// TIA Portal V19 export
TYPE "UDT_CONTROLVALVE"
   STRUCT
      pid : Struct   // PID
         mode { S7_SetPoint := 'True'} : Bool := false;   // Auto=0, Man=1
         action { S7_SetPoint := 'True'} : Bool := false;   // Reverse=0, Forward=1
         spsource : Bool := false;   // 0=internal setpoint, 1=external setpoint
         followup : Bool := false;   // 0=motor control from PID, 1=motor setpoint directly from program
         cmdrst : Bool := false;   // Controller reset command
         pidrun : Bool := false;   // Controller is running
         P { S7_SetPoint := 'True'} : Real := 0.0;   // Proportional gain
         I { S7_SetPoint := 'True'} : DInt := 0;   // Integral action
         D { S7_SetPoint := 'True'} : DInt := 0;   // Derivative action
         SP { S7_SetPoint := 'True'} : Real := 0.0;   // Setpoint
         PV : Real := 0.0;   // Peripheral value
         OFFVAL { S7_SetPoint := 'True'} : Real := 0.0;   // Value loaded to OP when the actuator is stopped
         LMN : Real := 0.0;   // Output of the PID controller
         OP { S7_SetPoint := 'True'} : Real := 0.0;   // Final output to the element
         L { S7_SetPoint := 'True'} : Real := 0.0;   // Lower value
         H { S7_SetPoint := 'True'} : Real := 0.0;   // Higher value
         EXT_SP : Real := 0.0;   // External setpoint
         FUP : Real := 0.0;   // Follow up value
         ITLVAL { S7_SetPoint := 'True'} : Real := 0.0;   // Controller initialization value
         pvunit { S7_SetPoint := 'True'} : WString := WSTRING#'';   // PV Unit
         outunit { S7_SetPoint := 'True'} : WString := WSTRING#'';   // Output Unit
         init : Struct   // Controller initialization routine
            req : Bool := false;   // An initialization routine is required
            dur { S7_SetPoint := 'True'} : Real := 0.0;   // Initialization duration
            delay : "UDT_DELAYON";
         END_STRUCT;
      END_STRUCT;
      unscale : Struct   // Scale output
         in : Real := 0.0;   // Value to be unscaled
         inhigh { S7_SetPoint := 'True'} : Real := 0.0;   // High limit of scale process (input value)
         inlow { S7_SetPoint := 'True'} : Real := 0.0;   // Low limit of scale process (input value)
         outhigh { S7_SetPoint := 'True'} : Real := 0.0;   // High limit of scale process (output value)
         outlow { S7_SetPoint := 'True'} : Real := 0.0;   // Low limit of scale process (output value)
         output : Real := 0.0;   // Unscaled value (only linear and span > 0)
         set : Bool := false;   // The scaling function is set
      END_STRUCT;
      status : Struct   // Status
         ilstart : Bool := false;   // Interlock start box
         icon : Int := 0;   // Valve icon
      END_STRUCT;
      out : Struct   // Output
         ref : Int := 0;   // Reference to control valve
         control : Bool := false;   // Command to start controlling
         vfbact : Bool := false;   // Virtual feedback "Open"
         vfbdeact : Bool := false;   // Virtual feedback "Close"
      END_STRUCT;
   END_STRUCT;
END_TYPE
